FUNCTION_BLOCK SENSOR_DETECTOR
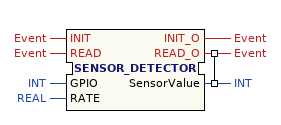
  EVENT_INPUT
    INIT;
    READ;
  END_EVENT
  EVENT_OUTPUT
    INIT_O;
    READ_O WITH SensorValue;
  END_EVENT
  VAR_INPUT
    GPIO : INT;
    RATE : REAL;
  END_VAR
  VAR_OUTPUT
    SensorValue : INT;
  END_VAR
END_FUNCTION_BLOCK
